(* Logix 5000 project; controller CarbonScout_MK6 vendor 1 type 14 code 154 rev 32.11; software revision 32.00; part 17 of 17 *)
(* tags used below, declared in another part *)
   ValveOneshot : DINT;
   CS_Alarms : P_Alarm[80];
   CS_Seq : GEK_Sequence;
   NetworkHealthy : DINT;
   Valve_SPR_01 : P_ValveSO;   // Air injection valve
   Valve_SPR_01_Stats : GekkoValveStat;
   Valve_XV_01 : P_ValveSO;   // Sample Valve Tank 1
   Valve_XV_01_Stats : GekkoValveStat;
   Valve_XV_02 : P_ValveSO;   // Sample Valve Tank 2
   Valve_XV_02_Stats : GekkoValveStat;
   Valve_XV_03 : P_ValveSO;   // Sample Valve Tank 3
   Valve_XV_03_Stats : GekkoValveStat;
   Valve_XV_04 : P_ValveSO;   // Sample Valve Tank 4
   Valve_XV_04_Stats : GekkoValveStat;
   Valve_XV_05 : P_ValveSO;   // Sample Valve Tank 5
   Valve_XV_05_Stats : GekkoValveStat;
   Valve_XV_06 : P_ValveSO;   // Sample Valve Tank 6
   Valve_XV_06_Stats : GekkoValveStat;
   Valve_XV_07 : P_ValveSO;   // Sample Valve Tank 7
   Valve_XV_07_Stats : GekkoValveStat;
   Valve_XV_08 : P_ValveSO;   // Sample Valve Tank 8
   Valve_XV_08_Stats : GekkoValveStat;
   Valve_XV_09 : P_ValveSO;   // Sample Valve Tank 9
   Valve_XV_09_Stats : GekkoValveStat;
   Valve_XV_10 : P_ValveSO;   // Sample Valve Tank 10
   Valve_XV_10_Stats : GekkoValveStat;
   Valve_XV_11 : P_ValveSO;   // Purge Valve
   Valve_XV_11_Stats : GekkoValveStat;
   Valve_XV_12 : P_ValveSO;   // Slurry inlet vavle
   Valve_XV_12_Stats : GekkoValveStat;
   Valve_XV_13 : P_ValveSO;   // Sample line vavle
   Valve_XV_13_Stats : GekkoValveStat;
   Valve_XV_14 : P_ValveSO;   // Top wash vavle
   Valve_XV_14_Stats : GekkoValveStat;
   Valve_XV_15 : P_ValveSO;   // Bottme wash vavle
   Valve_XV_15_Stats : GekkoValveStat;
   Valve_XV_16 : P_ValveSO;   // Potable water valve / Supply Water Valve
   Valve_XV_16_Stats : GekkoValveStat;
   Valve_XV_17 : P_ValveSO;   // Sample cone outlet vavle
   Valve_XV_17_Stats : GekkoValveStat;
   Valve_XV_18 : P_ValveSO;   // Sample strainer discharge
   Valve_XV_18_Stats : GekkoValveStat;
   Valve_XV_19 : P_ValveSO;   // Laser window
   Valve_XV_19_Stats : GekkoValveStat;
   Valve_XV_21_30 : P_ValveSO;   // Sample isolation valve
   Valve_XV_21_30_Stats : GekkoValveStat;
   Valve_XV_30 : P_ValveSO;   // XRF cooling valve
   Valve_XV_30_Stats : GekkoValveStat;
   Valve_XV_40 : P_ValveSO;   // XRF power on valve
(* Valves, continued *)

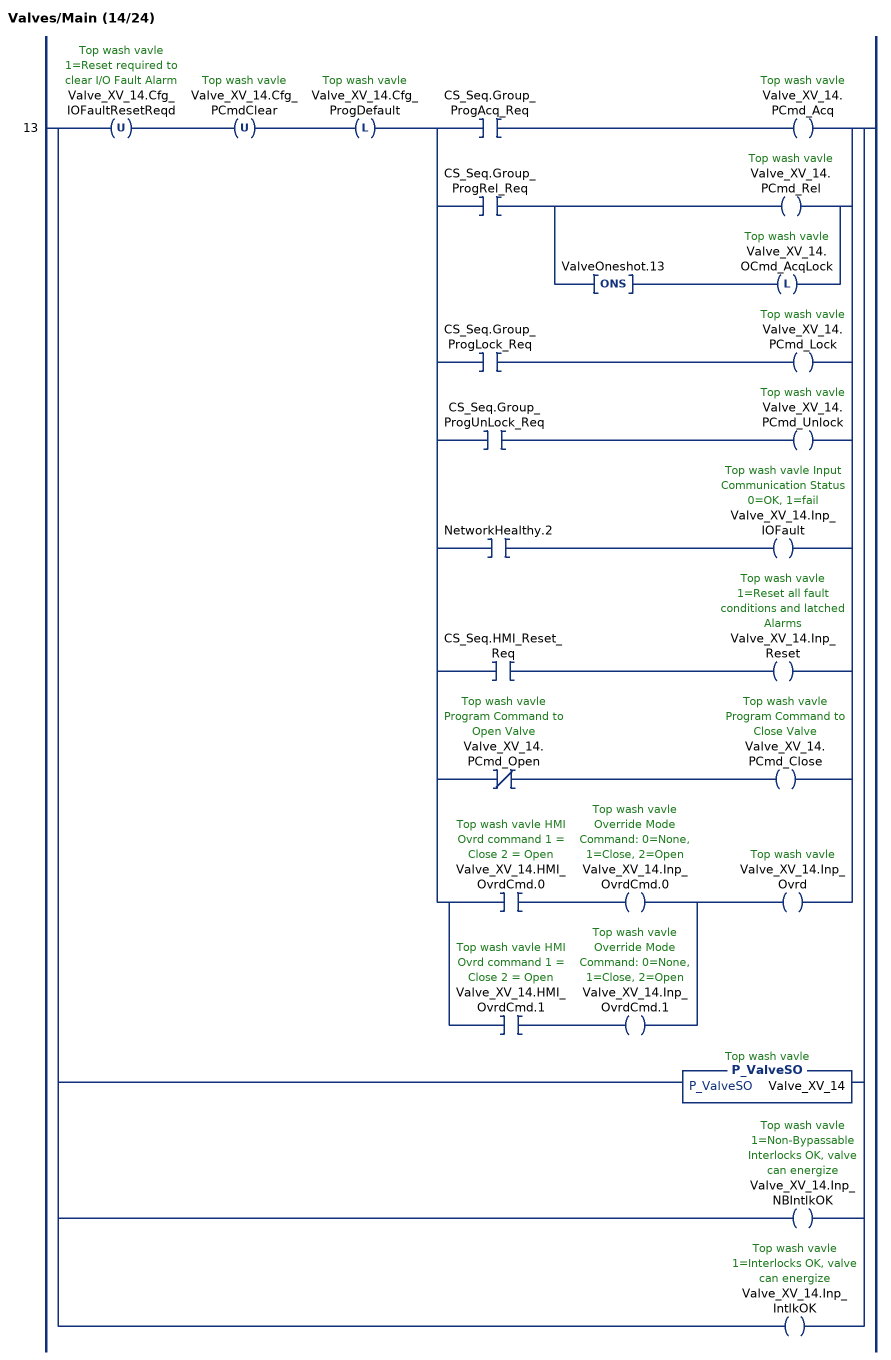
   [picture p361: Valves/Main rungs 13-13]
   13: [OTU(Valve_XV_14.Cfg_IOFaultResetReqd) OTU(Valve_XV_14.Cfg_PCmdClear) OTL(Valve_XV_14.Cfg_ProgDefault) [XIC(CS_Seq.Group_ProgAcq_Req) OTE(Valve_XV_14.PCmd_Acq) ,XIC(CS_Seq.Group_ProgRel_Req) [OTE(Valve_XV_14.PCmd_Rel) ,ONS(ValveOneshot.13) OTL(Valve_XV_14.OCmd_AcqLock) ] ,XIC(CS_Seq.Group_ProgLock_Req) OTE(Valve_XV_14.PCmd_Lock) ,XIC(CS_Seq.Group_ProgUnLock_Req) OTE(Valve_XV_14.PCmd_Unlock) ,XIC(NetworkHealthy.2) OTE(Valve_XV_14.Inp_IOFault) ,XIC(CS_Seq.HMI_Reset_Req) OTE(Valve_XV_14.Inp_Reset) ,XIO(Valve_XV_14.PCmd_Open) OTE(Valve_XV_14.PCmd_Close) ,[XIC(Valve_XV_14.HMI_OvrdCmd.0) OTE(Valve_XV_14.Inp_OvrdCmd.0) ,XIC(Valve_XV_14.HMI_OvrdCmd.1) OTE(Valve_XV_14.Inp_OvrdCmd.1) ] OTE(Valve_XV_14.Inp_Ovrd) ] ,[P_ValveSO(Valve_XV_14) ,OTE(Valve_XV_14.Inp_NBIntlkOK) ,OTE(Valve_XV_14.Inp_IntlkOK) ] ];
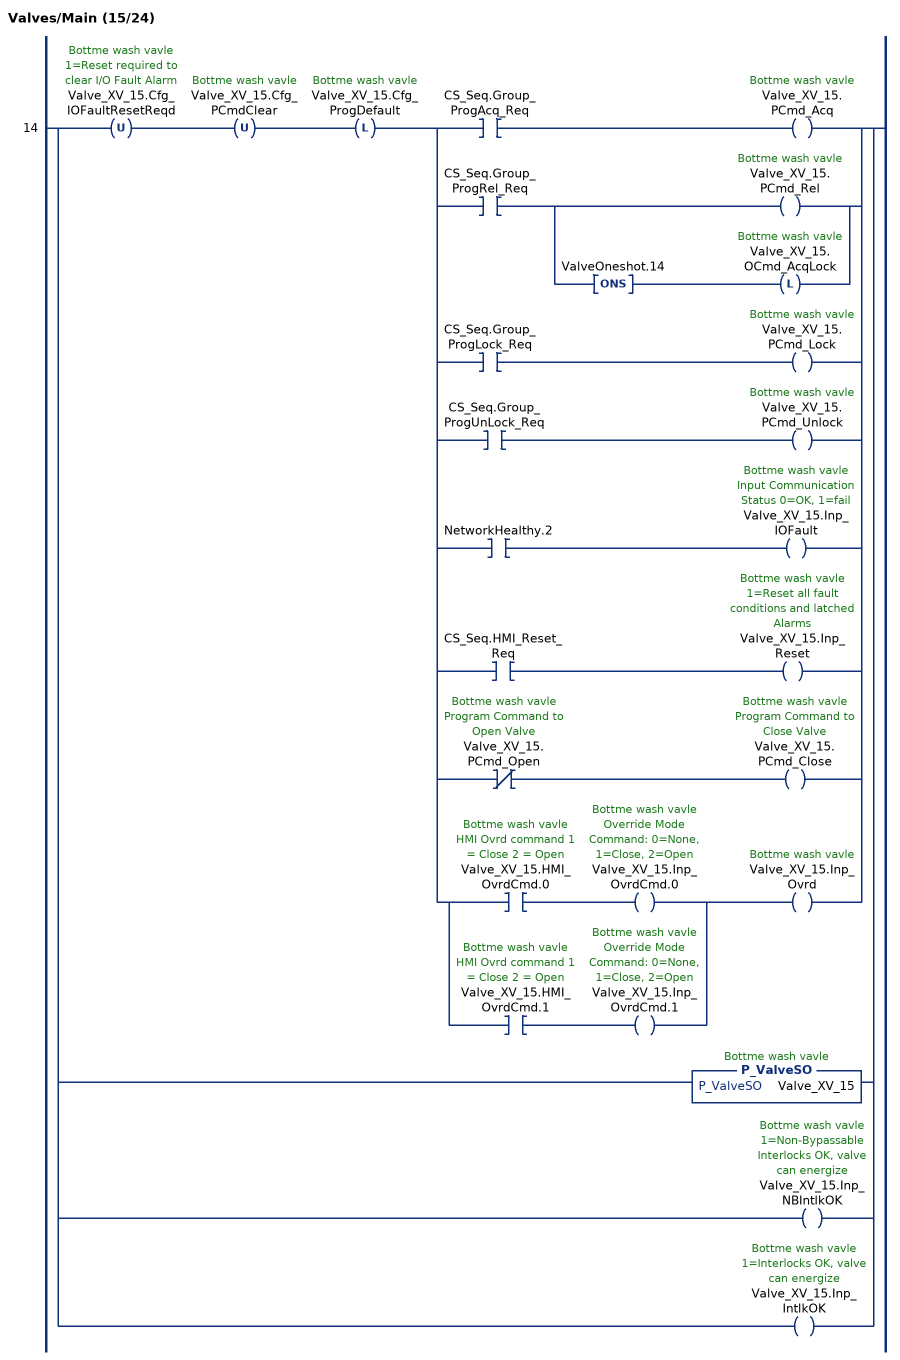
   14: [OTU(Valve_XV_15.Cfg_IOFaultResetReqd) OTU(Valve_XV_15.Cfg_PCmdClear) OTL(Valve_XV_15.Cfg_ProgDefault) [XIC(CS_Seq.Group_ProgAcq_Req) OTE(Valve_XV_15.PCmd_Acq) ,XIC(CS_Seq.Group_ProgRel_Req) [OTE(Valve_XV_15.PCmd_Rel) ,ONS(ValveOneshot.14) OTL(Valve_XV_15.OCmd_AcqLock) ] ,XIC(CS_Seq.Group_ProgLock_Req) OTE(Valve_XV_15.PCmd_Lock) ,XIC(CS_Seq.Group_ProgUnLock_Req) OTE(Valve_XV_15.PCmd_Unlock) ,XIC(NetworkHealthy.2) OTE(Valve_XV_15.Inp_IOFault) ,XIC(CS_Seq.HMI_Reset_Req) OTE(Valve_XV_15.Inp_Reset) ,XIO(Valve_XV_15.PCmd_Open) OTE(Valve_XV_15.PCmd_Close) ,[XIC(Valve_XV_15.HMI_OvrdCmd.0) OTE(Valve_XV_15.Inp_OvrdCmd.0) ,XIC(Valve_XV_15.HMI_OvrdCmd.1) OTE(Valve_XV_15.Inp_OvrdCmd.1) ] OTE(Valve_XV_15.Inp_Ovrd) ] ,[P_ValveSO(Valve_XV_15) ,OTE(Valve_XV_15.Inp_NBIntlkOK) ,OTE(Valve_XV_15.Inp_IntlkOK) ] ];
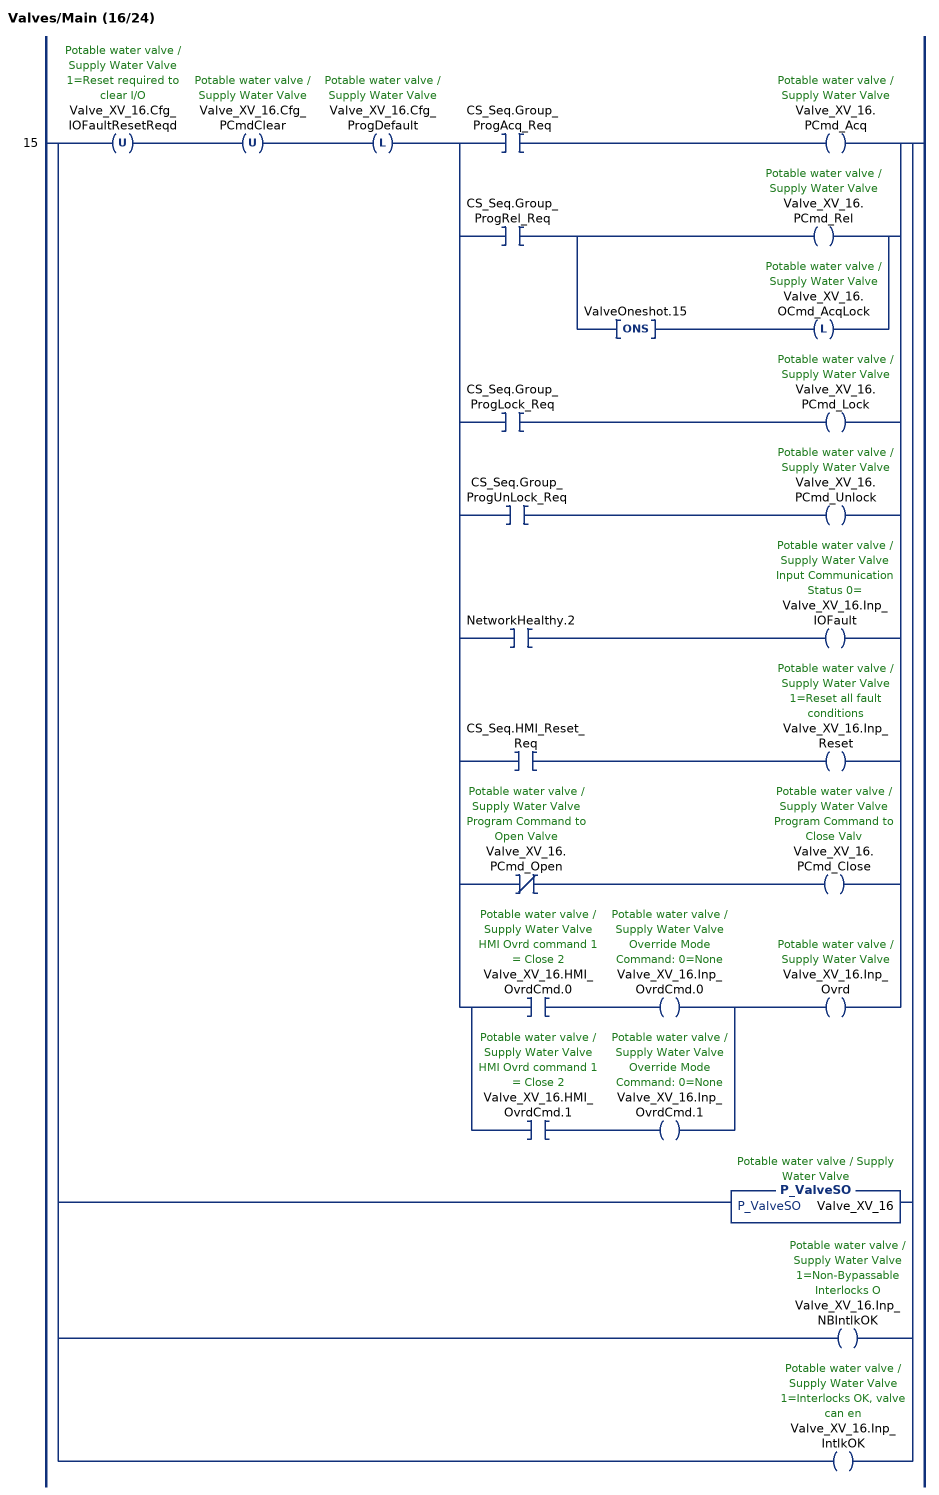
   15: [OTU(Valve_XV_16.Cfg_IOFaultResetReqd) OTU(Valve_XV_16.Cfg_PCmdClear) OTL(Valve_XV_16.Cfg_ProgDefault) [XIC(CS_Seq.Group_ProgAcq_Req) OTE(Valve_XV_16.PCmd_Acq) ,XIC(CS_Seq.Group_ProgRel_Req) [OTE(Valve_XV_16.PCmd_Rel) ,ONS(ValveOneshot.15) OTL(Valve_XV_16.OCmd_AcqLock) ] ,XIC(CS_Seq.Group_ProgLock_Req) OTE(Valve_XV_16.PCmd_Lock) ,XIC(CS_Seq.Group_ProgUnLock_Req) OTE(Valve_XV_16.PCmd_Unlock) ,XIC(NetworkHealthy.2) OTE(Valve_XV_16.Inp_IOFault) ,XIC(CS_Seq.HMI_Reset_Req) OTE(Valve_XV_16.Inp_Reset) ,XIO(Valve_XV_16.PCmd_Open) OTE(Valve_XV_16.PCmd_Close) ,[XIC(Valve_XV_16.HMI_OvrdCmd.0) OTE(Valve_XV_16.Inp_OvrdCmd.0) ,XIC(Valve_XV_16.HMI_OvrdCmd.1) OTE(Valve_XV_16.Inp_OvrdCmd.1) ] OTE(Valve_XV_16.Inp_Ovrd) ] ,[P_ValveSO(Valve_XV_16) ,OTE(Valve_XV_16.Inp_NBIntlkOK) ,OTE(Valve_XV_16.Inp_IntlkOK) ] ];
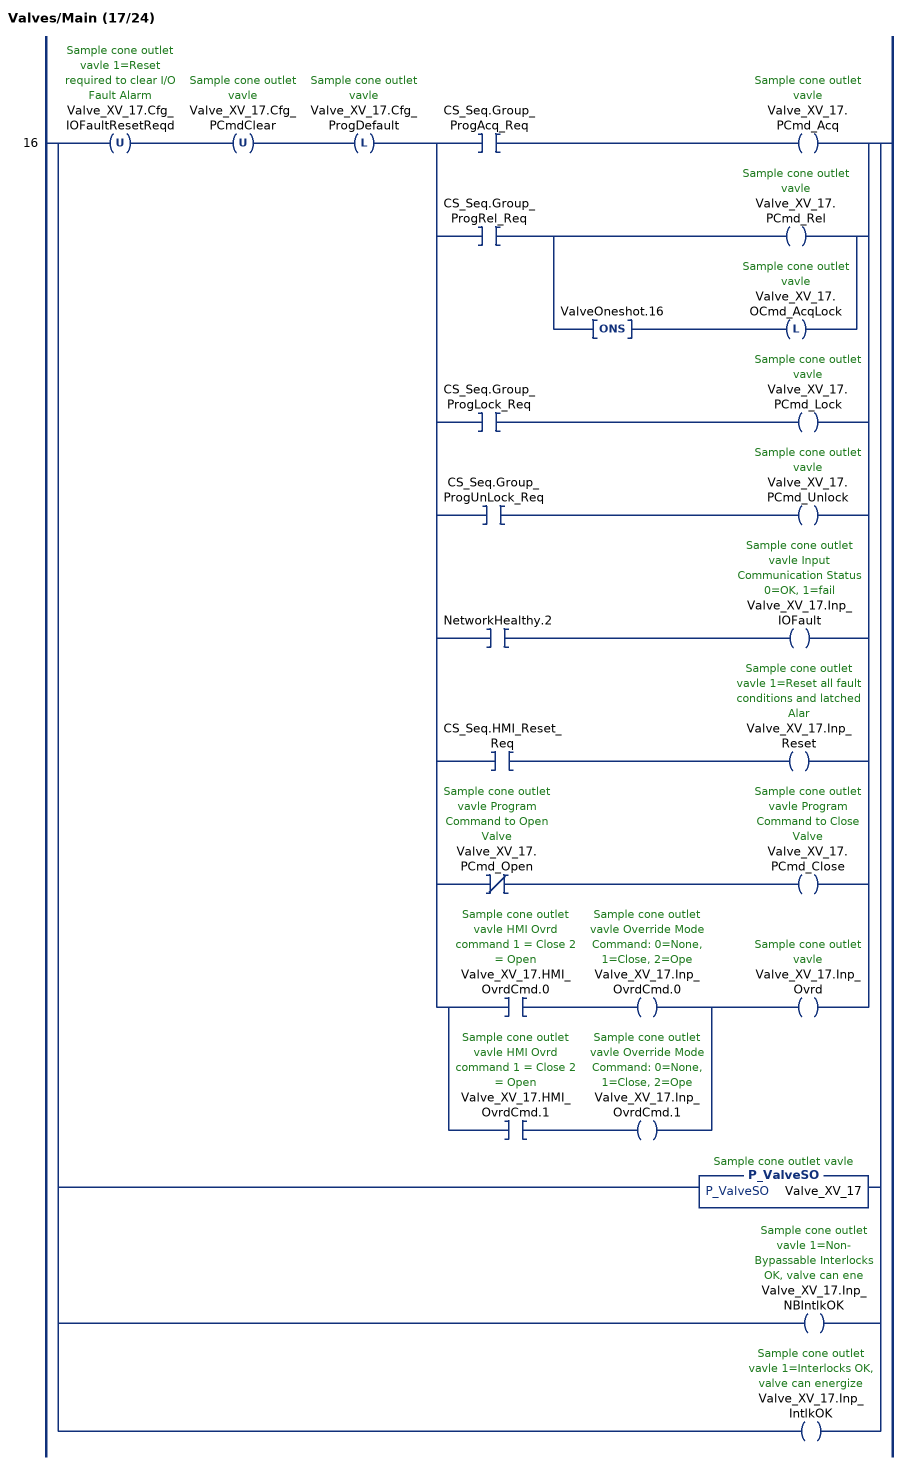
   16: [OTU(Valve_XV_17.Cfg_IOFaultResetReqd) OTU(Valve_XV_17.Cfg_PCmdClear) OTL(Valve_XV_17.Cfg_ProgDefault) [XIC(CS_Seq.Group_ProgAcq_Req) OTE(Valve_XV_17.PCmd_Acq) ,XIC(CS_Seq.Group_ProgRel_Req) [OTE(Valve_XV_17.PCmd_Rel) ,ONS(ValveOneshot.16) OTL(Valve_XV_17.OCmd_AcqLock) ] ,XIC(CS_Seq.Group_ProgLock_Req) OTE(Valve_XV_17.PCmd_Lock) ,XIC(CS_Seq.Group_ProgUnLock_Req) OTE(Valve_XV_17.PCmd_Unlock) ,XIC(NetworkHealthy.2) OTE(Valve_XV_17.Inp_IOFault) ,XIC(CS_Seq.HMI_Reset_Req) OTE(Valve_XV_17.Inp_Reset) ,XIO(Valve_XV_17.PCmd_Open) OTE(Valve_XV_17.PCmd_Close) ,[XIC(Valve_XV_17.HMI_OvrdCmd.0) OTE(Valve_XV_17.Inp_OvrdCmd.0) ,XIC(Valve_XV_17.HMI_OvrdCmd.1) OTE(Valve_XV_17.Inp_OvrdCmd.1) ] OTE(Valve_XV_17.Inp_Ovrd) ] ,[P_ValveSO(Valve_XV_17) ,OTE(Valve_XV_17.Inp_NBIntlkOK) ,OTE(Valve_XV_17.Inp_IntlkOK) ] ];
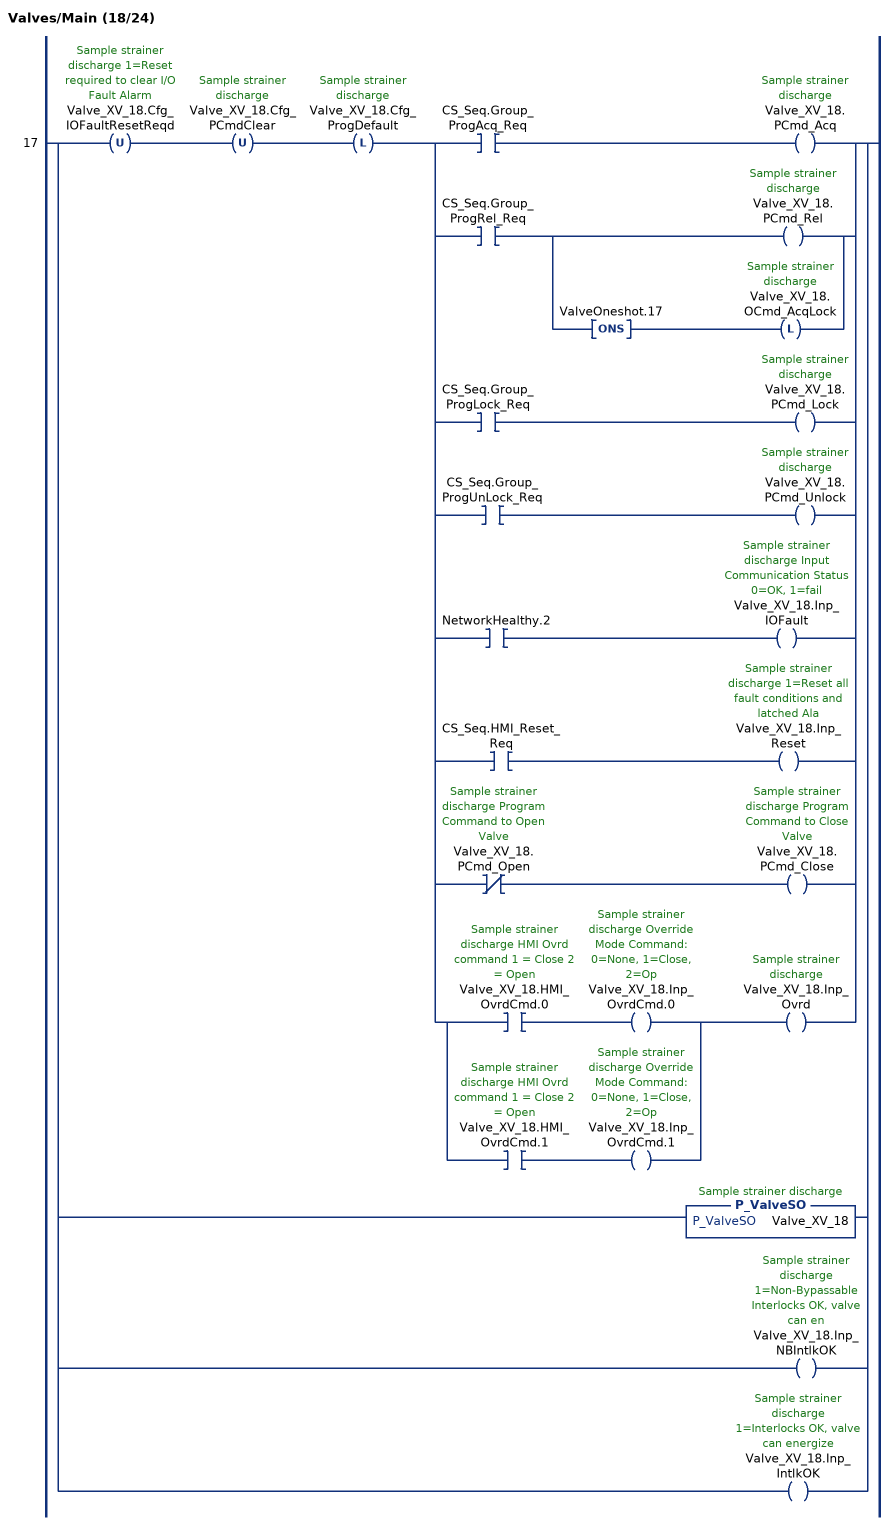
   17: [OTU(Valve_XV_18.Cfg_IOFaultResetReqd) OTU(Valve_XV_18.Cfg_PCmdClear) OTL(Valve_XV_18.Cfg_ProgDefault) [XIC(CS_Seq.Group_ProgAcq_Req) OTE(Valve_XV_18.PCmd_Acq) ,XIC(CS_Seq.Group_ProgRel_Req) [OTE(Valve_XV_18.PCmd_Rel) ,ONS(ValveOneshot.17) OTL(Valve_XV_18.OCmd_AcqLock) ] ,XIC(CS_Seq.Group_ProgLock_Req) OTE(Valve_XV_18.PCmd_Lock) ,XIC(CS_Seq.Group_ProgUnLock_Req) OTE(Valve_XV_18.PCmd_Unlock) ,XIC(NetworkHealthy.2) OTE(Valve_XV_18.Inp_IOFault) ,XIC(CS_Seq.HMI_Reset_Req) OTE(Valve_XV_18.Inp_Reset) ,XIO(Valve_XV_18.PCmd_Open) OTE(Valve_XV_18.PCmd_Close) ,[XIC(Valve_XV_18.HMI_OvrdCmd.0) OTE(Valve_XV_18.Inp_OvrdCmd.0) ,XIC(Valve_XV_18.HMI_OvrdCmd.1) OTE(Valve_XV_18.Inp_OvrdCmd.1) ] OTE(Valve_XV_18.Inp_Ovrd) ] ,[P_ValveSO(Valve_XV_18) ,OTE(Valve_XV_18.Inp_NBIntlkOK) ,OTE(Valve_XV_18.Inp_IntlkOK) ] ];
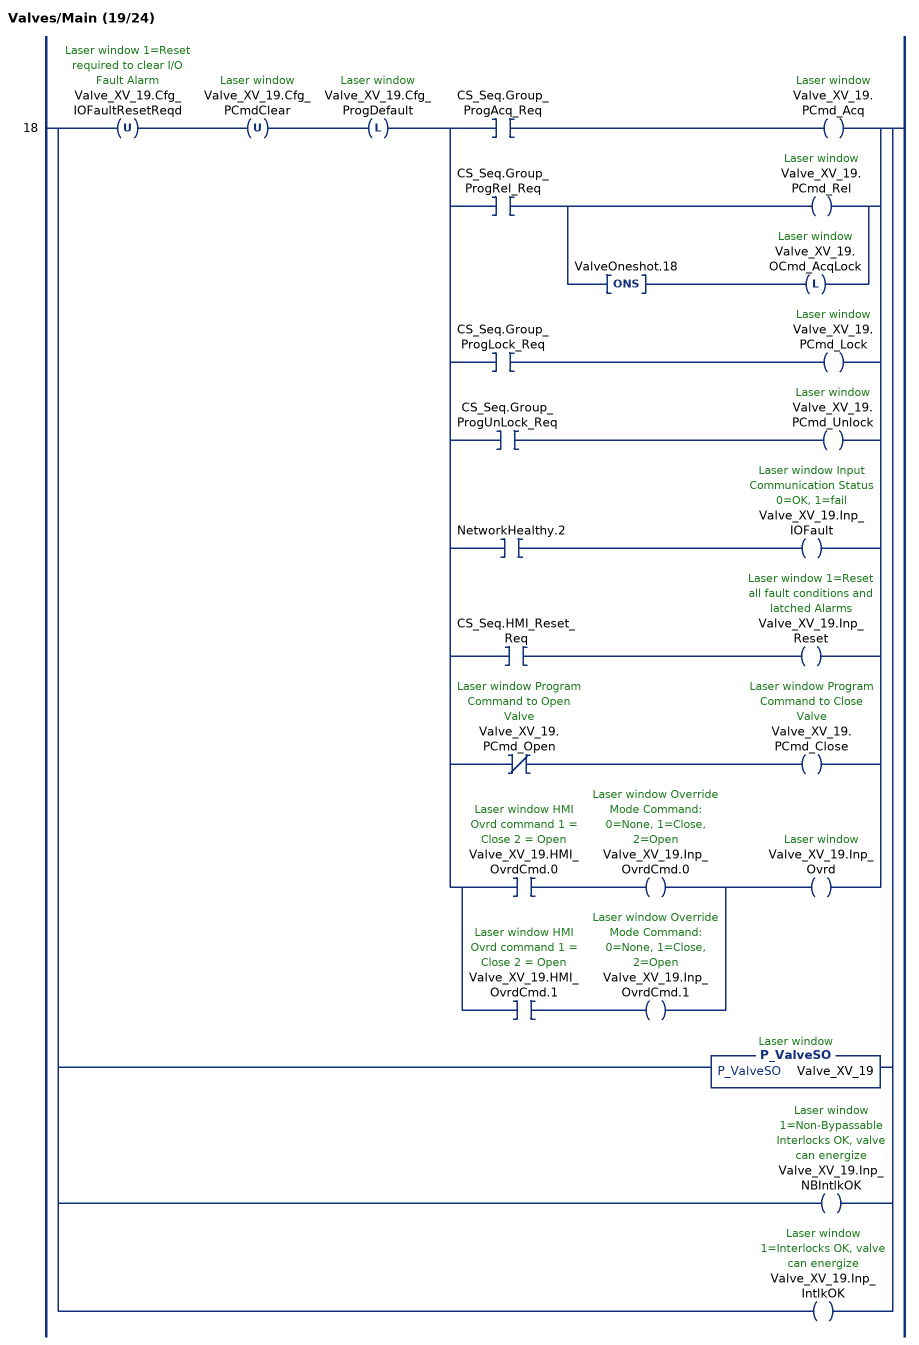
   18: [OTU(Valve_XV_19.Cfg_IOFaultResetReqd) OTU(Valve_XV_19.Cfg_PCmdClear) OTL(Valve_XV_19.Cfg_ProgDefault) [XIC(CS_Seq.Group_ProgAcq_Req) OTE(Valve_XV_19.PCmd_Acq) ,XIC(CS_Seq.Group_ProgRel_Req) [OTE(Valve_XV_19.PCmd_Rel) ,ONS(ValveOneshot.18) OTL(Valve_XV_19.OCmd_AcqLock) ] ,XIC(CS_Seq.Group_ProgLock_Req) OTE(Valve_XV_19.PCmd_Lock) ,XIC(CS_Seq.Group_ProgUnLock_Req) OTE(Valve_XV_19.PCmd_Unlock) ,XIC(NetworkHealthy.2) OTE(Valve_XV_19.Inp_IOFault) ,XIC(CS_Seq.HMI_Reset_Req) OTE(Valve_XV_19.Inp_Reset) ,XIO(Valve_XV_19.PCmd_Open) OTE(Valve_XV_19.PCmd_Close) ,[XIC(Valve_XV_19.HMI_OvrdCmd.0) OTE(Valve_XV_19.Inp_OvrdCmd.0) ,XIC(Valve_XV_19.HMI_OvrdCmd.1) OTE(Valve_XV_19.Inp_OvrdCmd.1) ] OTE(Valve_XV_19.Inp_Ovrd) ] ,[P_ValveSO(Valve_XV_19) ,OTE(Valve_XV_19.Inp_NBIntlkOK) ,OTE(Valve_XV_19.Inp_IntlkOK) ] ];
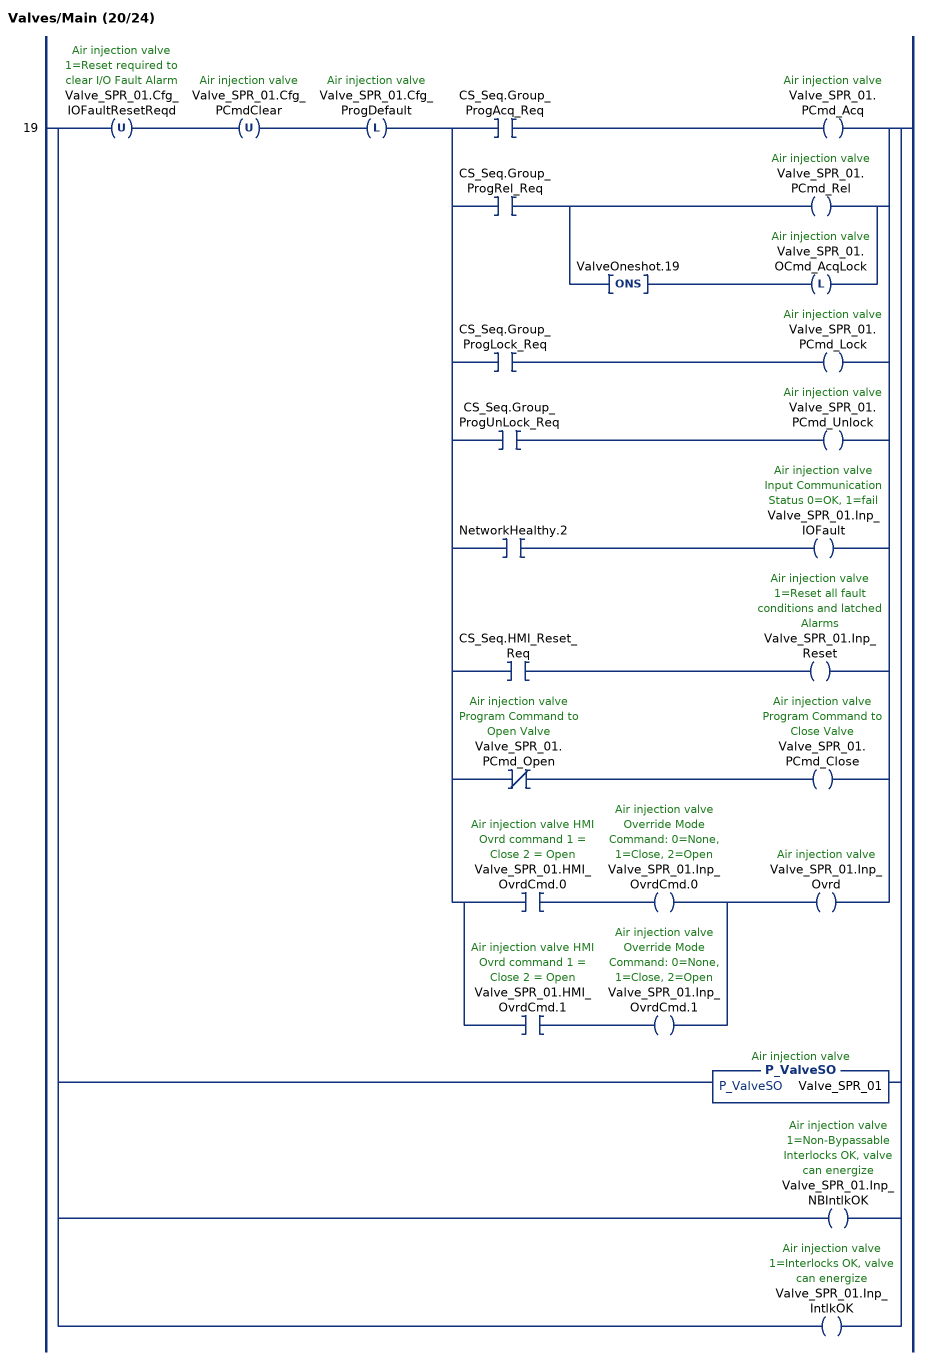
   19: [OTU(Valve_SPR_01.Cfg_IOFaultResetReqd) OTU(Valve_SPR_01.Cfg_PCmdClear) OTL(Valve_SPR_01.Cfg_ProgDefault) [XIC(CS_Seq.Group_ProgAcq_Req) OTE(Valve_SPR_01.PCmd_Acq) ,XIC(CS_Seq.Group_ProgRel_Req) [OTE(Valve_SPR_01.PCmd_Rel) ,ONS(ValveOneshot.19) OTL(Valve_SPR_01.OCmd_AcqLock) ] ,XIC(CS_Seq.Group_ProgLock_Req) OTE(Valve_SPR_01.PCmd_Lock) ,XIC(CS_Seq.Group_ProgUnLock_Req) OTE(Valve_SPR_01.PCmd_Unlock) ,XIC(NetworkHealthy.2) OTE(Valve_SPR_01.Inp_IOFault) ,XIC(CS_Seq.HMI_Reset_Req) OTE(Valve_SPR_01.Inp_Reset) ,XIO(Valve_SPR_01.PCmd_Open) OTE(Valve_SPR_01.PCmd_Close) ,[XIC(Valve_SPR_01.HMI_OvrdCmd.0) OTE(Valve_SPR_01.Inp_OvrdCmd.0) ,XIC(Valve_SPR_01.HMI_OvrdCmd.1) OTE(Valve_SPR_01.Inp_OvrdCmd.1) ] OTE(Valve_SPR_01.Inp_Ovrd) ] ,[P_ValveSO(Valve_SPR_01) ,OTE(Valve_SPR_01.Inp_NBIntlkOK) ,OTE(Valve_SPR_01.Inp_IntlkOK) ] ];
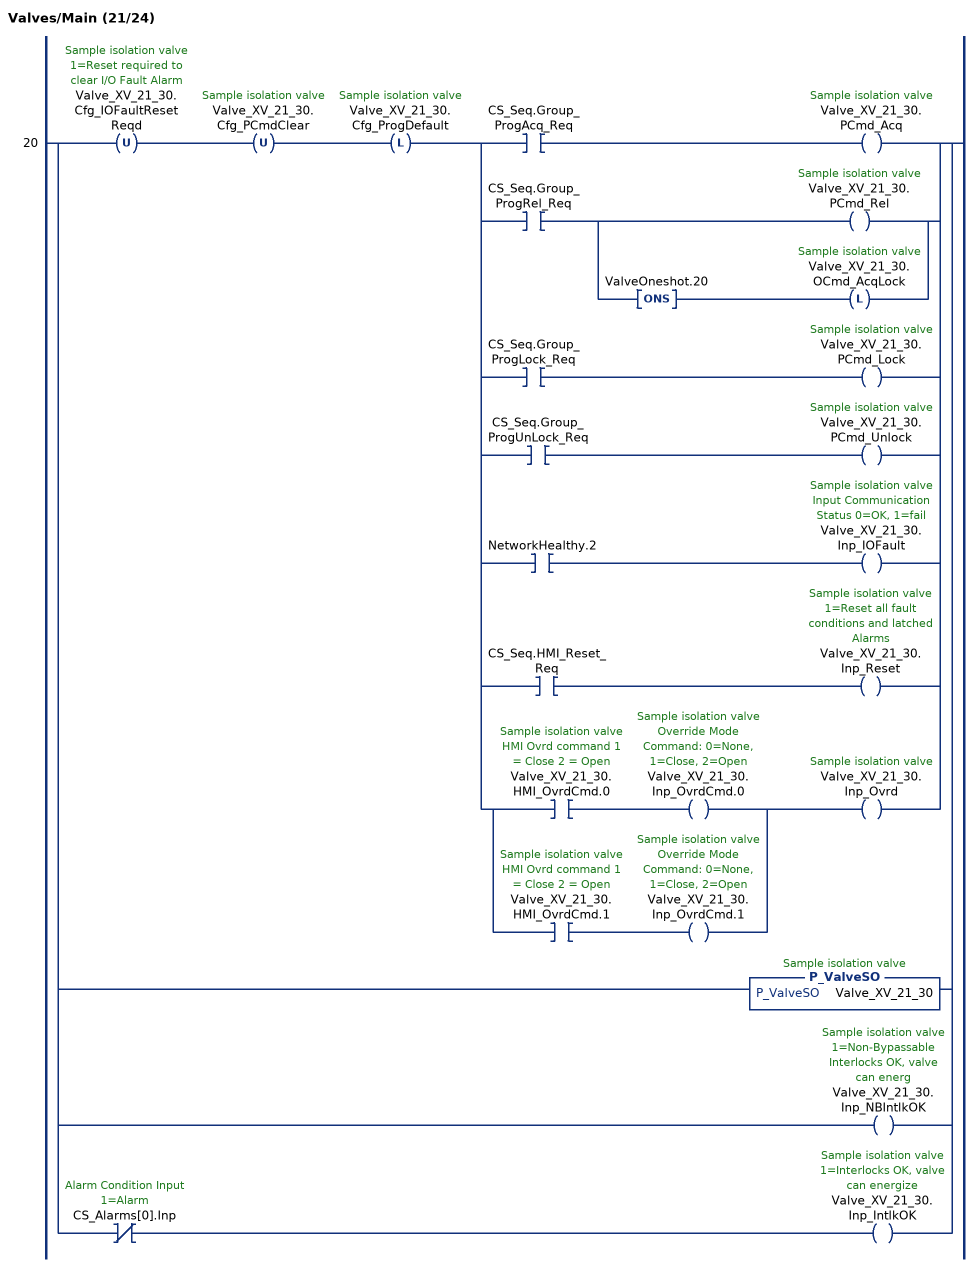
   20: [OTU(Valve_XV_21_30.Cfg_IOFaultResetReqd) OTU(Valve_XV_21_30.Cfg_PCmdClear) OTL(Valve_XV_21_30.Cfg_ProgDefault) [XIC(CS_Seq.Group_ProgAcq_Req) OTE(Valve_XV_21_30.PCmd_Acq) ,XIC(CS_Seq.Group_ProgRel_Req) [OTE(Valve_XV_21_30.PCmd_Rel) ,ONS(ValveOneshot.20) OTL(Valve_XV_21_30.OCmd_AcqLock) ] ,XIC(CS_Seq.Group_ProgLock_Req) OTE(Valve_XV_21_30.PCmd_Lock) ,XIC(CS_Seq.Group_ProgUnLock_Req) OTE(Valve_XV_21_30.PCmd_Unlock) ,XIC(NetworkHealthy.2) OTE(Valve_XV_21_30.Inp_IOFault) ,XIC(CS_Seq.HMI_Reset_Req) OTE(Valve_XV_21_30.Inp_Reset) ,[XIC(Valve_XV_21_30.HMI_OvrdCmd.0) OTE(Valve_XV_21_30.Inp_OvrdCmd.0) ,XIC(Valve_XV_21_30.HMI_OvrdCmd.1) OTE(Valve_XV_21_30.Inp_OvrdCmd.1) ] OTE(Valve_XV_21_30.Inp_Ovrd) ] ,[P_ValveSO(Valve_XV_21_30) ,OTE(Valve_XV_21_30.Inp_NBIntlkOK) ,XIO(CS_Alarms[0].Inp) OTE(Valve_XV_21_30.Inp_IntlkOK) ] ];
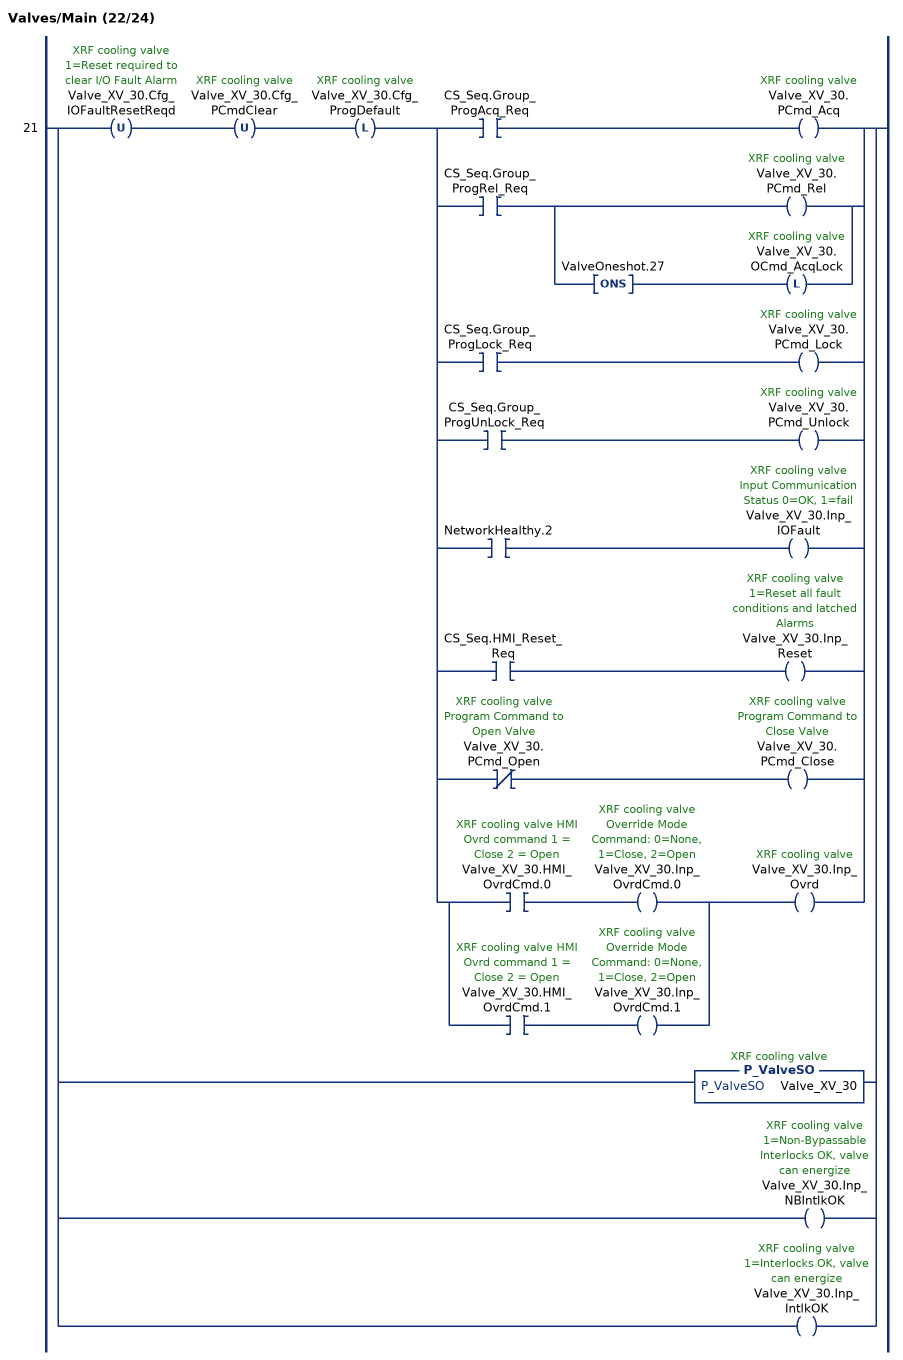
   21: [OTU(Valve_XV_30.Cfg_IOFaultResetReqd) OTU(Valve_XV_30.Cfg_PCmdClear) OTL(Valve_XV_30.Cfg_ProgDefault) [XIC(CS_Seq.Group_ProgAcq_Req) OTE(Valve_XV_30.PCmd_Acq) ,XIC(CS_Seq.Group_ProgRel_Req) [OTE(Valve_XV_30.PCmd_Rel) ,ONS(ValveOneshot.27) OTL(Valve_XV_30.OCmd_AcqLock) ] ,XIC(CS_Seq.Group_ProgLock_Req) OTE(Valve_XV_30.PCmd_Lock) ,XIC(CS_Seq.Group_ProgUnLock_Req) OTE(Valve_XV_30.PCmd_Unlock) ,XIC(NetworkHealthy.2) OTE(Valve_XV_30.Inp_IOFault) ,XIC(CS_Seq.HMI_Reset_Req) OTE(Valve_XV_30.Inp_Reset) ,XIO(Valve_XV_30.PCmd_Open) OTE(Valve_XV_30.PCmd_Close) ,[XIC(Valve_XV_30.HMI_OvrdCmd.0) OTE(Valve_XV_30.Inp_OvrdCmd.0) ,XIC(Valve_XV_30.HMI_OvrdCmd.1) OTE(Valve_XV_30.Inp_OvrdCmd.1) ] OTE(Valve_XV_30.Inp_Ovrd) ] ,[P_ValveSO(Valve_XV_30) ,OTE(Valve_XV_30.Inp_NBIntlkOK) ,OTE(Valve_XV_30.Inp_IntlkOK) ] ];
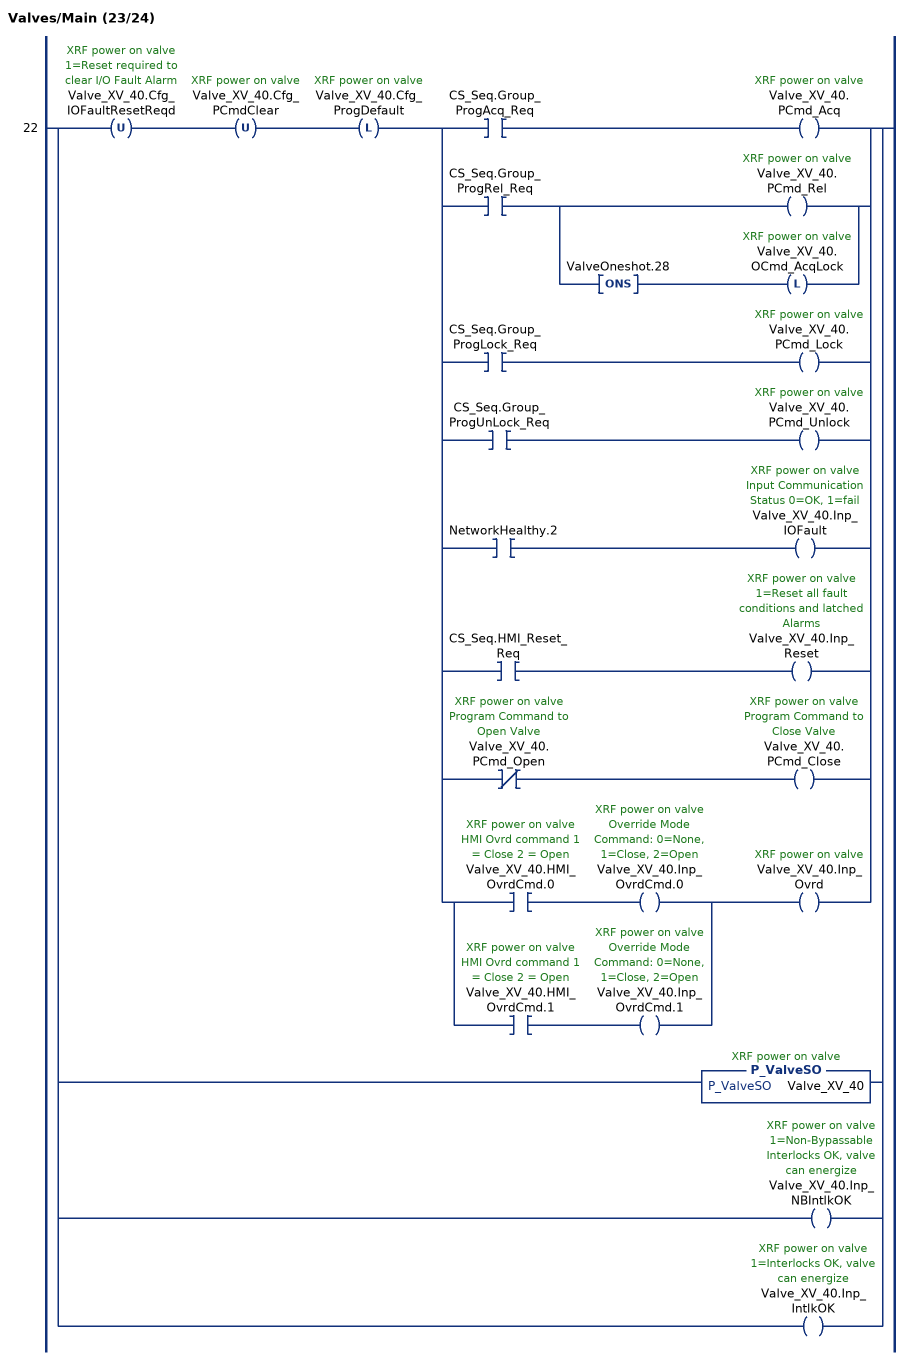
   22: [OTU(Valve_XV_40.Cfg_IOFaultResetReqd) OTU(Valve_XV_40.Cfg_PCmdClear) OTL(Valve_XV_40.Cfg_ProgDefault) [XIC(CS_Seq.Group_ProgAcq_Req) OTE(Valve_XV_40.PCmd_Acq) ,XIC(CS_Seq.Group_ProgRel_Req) [OTE(Valve_XV_40.PCmd_Rel) ,ONS(ValveOneshot.28) OTL(Valve_XV_40.OCmd_AcqLock) ] ,XIC(CS_Seq.Group_ProgLock_Req) OTE(Valve_XV_40.PCmd_Lock) ,XIC(CS_Seq.Group_ProgUnLock_Req) OTE(Valve_XV_40.PCmd_Unlock) ,XIC(NetworkHealthy.2) OTE(Valve_XV_40.Inp_IOFault) ,XIC(CS_Seq.HMI_Reset_Req) OTE(Valve_XV_40.Inp_Reset) ,XIO(Valve_XV_40.PCmd_Open) OTE(Valve_XV_40.PCmd_Close) ,[XIC(Valve_XV_40.HMI_OvrdCmd.0) OTE(Valve_XV_40.Inp_OvrdCmd.0) ,XIC(Valve_XV_40.HMI_OvrdCmd.1) OTE(Valve_XV_40.Inp_OvrdCmd.1) ] OTE(Valve_XV_40.Inp_Ovrd) ] ,[P_ValveSO(Valve_XV_40) ,OTE(Valve_XV_40.Inp_NBIntlkOK) ,OTE(Valve_XV_40.Inp_IntlkOK) ] ];
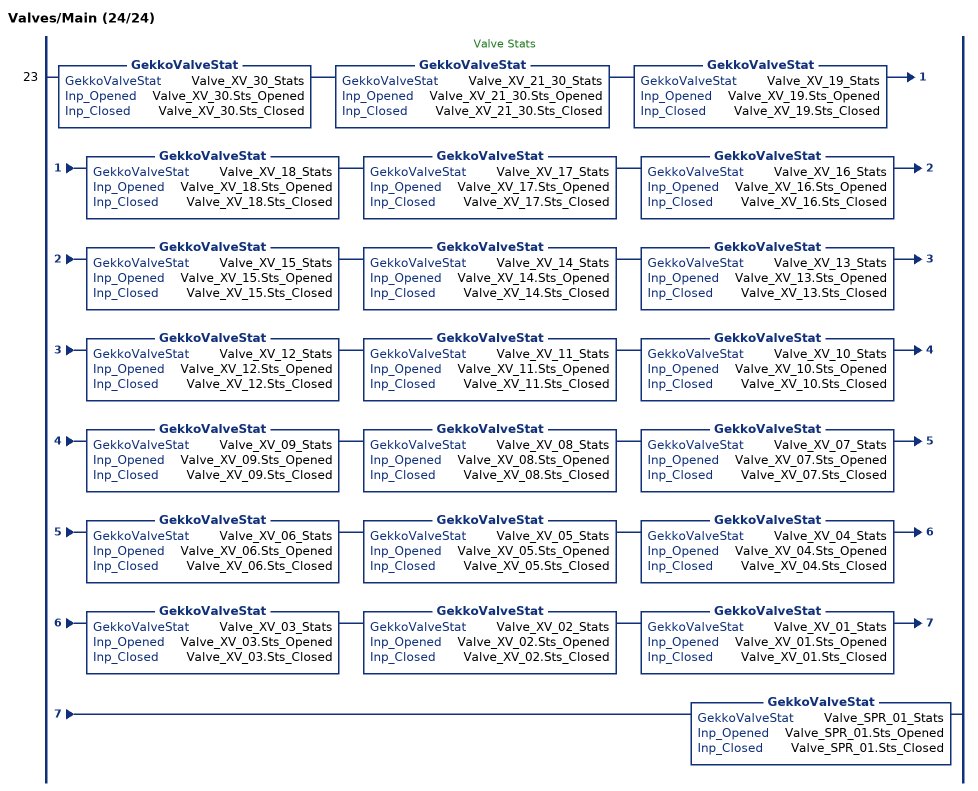
   // Valve Stats
   23: GekkoValveStat(Valve_XV_30_Stats,Valve_XV_30.Sts_Opened,Valve_XV_30.Sts_Closed)GekkoValveStat(Valve_XV_21_30_Stats,Valve_XV_21_30.Sts_Opened,Valve_XV_21_30.Sts_Closed)GekkoValveStat(Valve_XV_19_Stats,Valve_XV_19.Sts_Opened,Valve_XV_19.Sts_Closed)GekkoValveStat(Valve_XV_18_Stats,Valve_XV_18.Sts_Opened,Valve_XV_18.Sts_Closed)GekkoValveStat(Valve_XV_17_Stats,Valve_XV_17.Sts_Opened,Valve_XV_17.Sts_Closed)GekkoValveStat(Valve_XV_16_Stats,Valve_XV_16.Sts_Opened,Valve_XV_16.Sts_Closed)GekkoValveStat(Valve_XV_15_Stats,Valve_XV_15.Sts_Opened,Valve_XV_15.Sts_Closed)GekkoValveStat(Valve_XV_14_Stats,Valve_XV_14.Sts_Opened,Valve_XV_14.Sts_Closed)GekkoValveStat(Valve_XV_13_Stats,Valve_XV_13.Sts_Opened,Valve_XV_13.Sts_Closed)GekkoValveStat(Valve_XV_12_Stats,Valve_XV_12.Sts_Opened,Valve_XV_12.Sts_Closed)GekkoValveStat(Valve_XV_11_Stats,Valve_XV_11.Sts_Opened,Valve_XV_11.Sts_Closed)GekkoValveStat(Valve_XV_10_Stats,Valve_XV_10.Sts_Opened,Valve_XV_10.Sts_Closed)GekkoValveStat(Valve_XV_09_Stats,Valve_XV_09.Sts_Opened,Valve_XV_09.Sts_Closed)GekkoValveStat(Valve_XV_08_Stats,Valve_XV_08.Sts_Opened,Valve_XV_08.Sts_Closed)GekkoValveStat(Valve_XV_07_Stats,Valve_XV_07.Sts_Opened,Valve_XV_07.Sts_Closed)GekkoValveStat(Valve_XV_06_Stats,Valve_XV_06.Sts_Opened,Valve_XV_06.Sts_Closed)GekkoValveStat(Valve_XV_05_Stats,Valve_XV_05.Sts_Opened,Valve_XV_05.Sts_Closed)GekkoValveStat(Valve_XV_04_Stats,Valve_XV_04.Sts_Opened,Valve_XV_04.Sts_Closed)GekkoValveStat(Valve_XV_03_Stats,Valve_XV_03.Sts_Opened,Valve_XV_03.Sts_Closed)GekkoValveStat(Valve_XV_02_Stats,Valve_XV_02.Sts_Opened,Valve_XV_02.Sts_Closed)GekkoValveStat(Valve_XV_01_Stats,Valve_XV_01.Sts_Opened,Valve_XV_01.Sts_Closed)GekkoValveStat(Valve_SPR_01_Stats,Valve_SPR_01.Sts_Opened,Valve_SPR_01.Sts_Closed);
END_ROUTINE
END_PROGRAM
